(* This version of the block is self contained. Minimizes wiring.*)
FUNCTION_BLOCK FB_ExampleDeviceSM_DB
VAR_INPUT
	cBase: UDINT;
	iDBID:UDINT;
	sDBNetId: STRING;
	sDeviceID: STRING;
END_VAR
VAR_OUTPUT
END_VAR
VAR_IN_OUT
	fbArbiter : FB_Arbiter;
	fbFastFaultOutput	:	FB_HardwareFFOutput;
END_VAR
VAR
	stDevice	:	ST_Device;
	fbGovernor	:	FB_LinearGovernor;
	mcPower	:	MC_Power;
	mcStop: MC_Stop;
	mcAbsolute	:	MC_MoveAbsolute;
	fbBPTM	:	BeamParameterTransitionManager;
	xStartMove: BOOL;
	
	stCheckState: ST_DeviceState;
	stTargetState	:	ST_DeviceState; //Target device state
	fbDBClient:FB_MySQL_Client;
	bInitReady: BOOL :=FALSE;
	//aStateTable : ARRAY[1..PMPS_GVL.MAX_DEVICE_STATES] OF ST_DeviceStateTable;

END_VAR
VAR PERSISTENT
	nLastActiveState	:	UDINT;
END_VAR

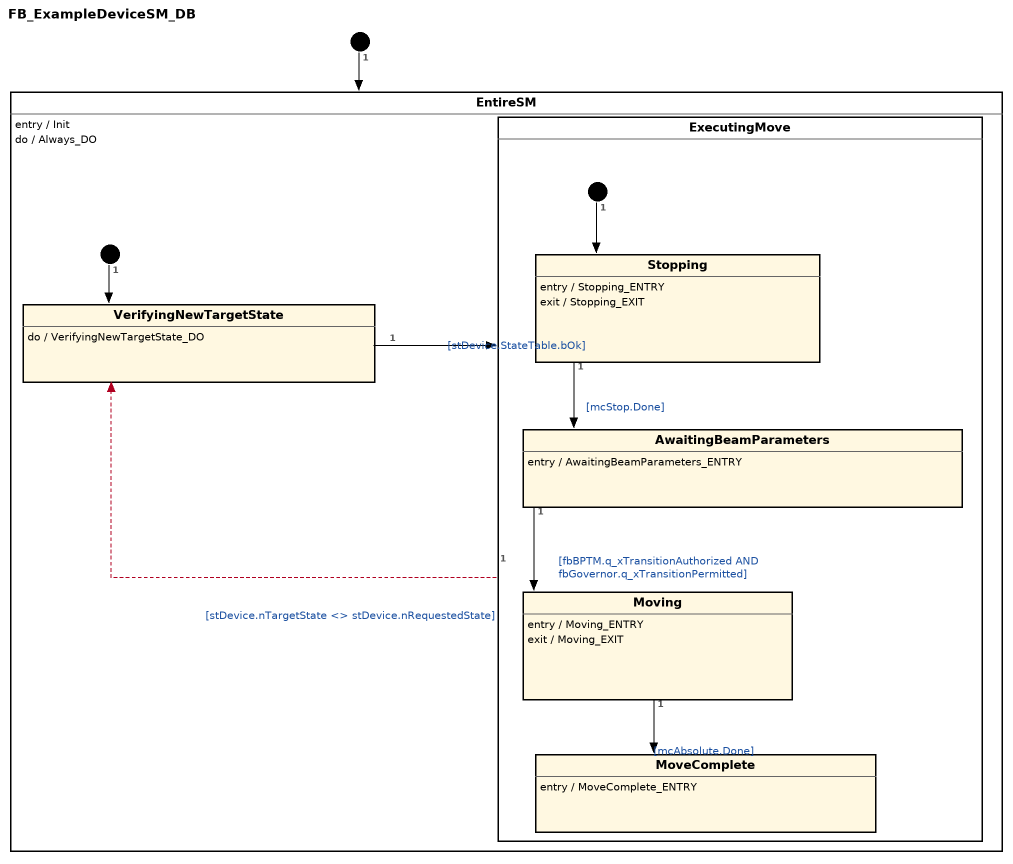
STATECHART FB_ExampleDeviceSM_DB  // abortable
    START StartState3
    COMPOSITE STATE EntireSM
        entry / Init
        do / Always_DO
        START StartState1
        COMPOSITE STATE ExecutingMove
            START StartState2
            STATE Stopping
                entry / Stopping_ENTRY
                exit / Stopping_EXIT
            STATE AwaitingBeamParameters
                entry / AwaitingBeamParameters_ENTRY
            STATE Moving
                entry / Moving_ENTRY
                exit / Moving_EXIT
            STATE MoveComplete
                entry / MoveComplete_ENTRY
            StartState2 -> Stopping  // priority 1, on completion
            Stopping -> AwaitingBeamParameters [mcStop.Done] // priority 1, rising edge
            AwaitingBeamParameters -> Moving [fbBPTM.q_xTransitionAuthorized AND fbGovernor.q_xTransitionPermitted] // priority 1, rising edge
            Moving -> MoveComplete [mcAbsolute.Done] // priority 1, rising edge
        END_STATE
        STATE VerifyingNewTargetState
            do / VerifyingNewTargetState_DO
        StartState1 -> VerifyingNewTargetState  // priority 1, on completion
        ExecutingMove -> VerifyingNewTargetState [stDevice.nTargetState <> stDevice.nRequestedState] // priority 1, exception, rising edge
        VerifyingNewTargetState -> ExecutingMove [stDevice.StateTable.bOk] // priority 1
    END_STATE
    StartState3 -> EntireSM  // priority 1, on completion
END_STATECHART

ACTION Always_DO:
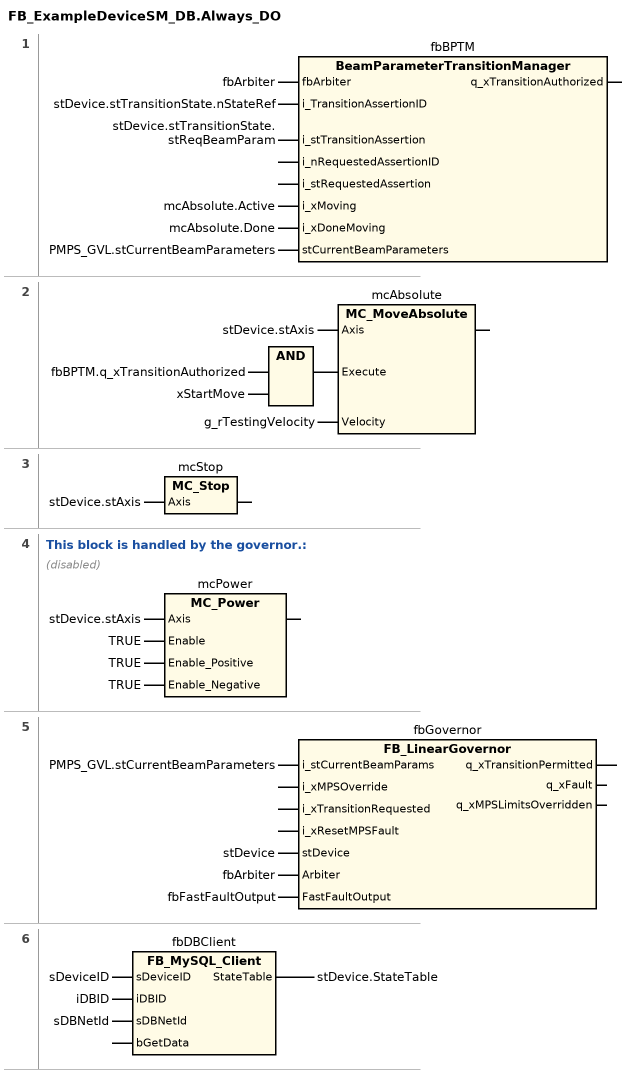
// NETWORK 1
fbBPTM(
    fbArbiter := fbArbiter,
    i_TransitionAssertionID := stDevice.stTransitionState.nStateRef,
    i_stTransitionAssertion := stDevice.stTransitionState.stReqBeamParam,
    i_xMoving := mcAbsolute.Active,
    i_xDoneMoving := mcAbsolute.Done,
    stCurrentBeamParameters := PMPS_GVL.stCurrentBeamParameters); // BeamParameterTransitionManager

// NETWORK 2
mcAbsolute(
    Axis := stDevice.stAxis,
    Execute := fbBPTM.q_xTransitionAuthorized AND xStartMove,
    Velocity := g_rTestingVelocity); // MC_MoveAbsolute

// NETWORK 3
mcStop(Axis := stDevice.stAxis); // MC_Stop

// NETWORK 4 (disabled)
// label: This block is handled by the governor.
// mcPower(Axis := stDevice.stAxis, Enable := TRUE, Enable_Positive := TRUE, Enable_Negative := TRUE); // MC_Power

// NETWORK 5
fbGovernor(
    i_stCurrentBeamParams := PMPS_GVL.stCurrentBeamParameters,
    stDevice := stDevice,
    Arbiter := fbArbiter,
    FastFaultOutput := fbFastFaultOutput); // FB_LinearGovernor

// NETWORK 6
fbDBClient(sDeviceID := sDeviceID, iDBID := iDBID, sDBNetId := sDBNetId); // FB_MySQL_Client
stDevice.StateTable := fbDBClient.StateTable;
END_ACTION

ACTION AwaitingBeamParameters_ENTRY:
fbBPTM.i_stRequestedAssertion := stTargetState.stReqBeamParam;
fbBPTM.i_nRequestedAssertionID := stTargetState.nStateRef;

//Tell the governor that we're trying to move.
fbGovernor.i_xTransitionRequested := TRUE;
END_ACTION

ACTION Init:
	
//Safe State
stDevice.nSafeState := cBase;
stDevice.nTransitionState := cBase+100;

//Initialize the State Table
stDevice.StateTable.A_Reset();
//Device State Table Instantiation
F_SetStateParams(
	nStateRef := stDevice.nSafeState,
	rPosition := 0,
	rTolerance := 10,
	stBeamParams := PMPS_GVL.cstFullBeam,
	Table := stDevice.StateTable
);
//Connect to DB and get state table data
fbDBClient.bGetData:= TRUE;//fbMySQL.nState:=400; 

stDevice.StateTable.A_Lookup(
		key := stDevice.nTransitionState,
		getValue => stDevice.stTransitionState
);
	
//Need an initialization routine for setting the active state
//Check if the device is at the last known state
//If the device is within the state boundaries, it's considered to be in that state
stDevice.StateTable.A_Lookup(key:= nLastActiveState);
IF stDevice.StateTable.bOk THEN
	stCheckState := stDevice.StateTable.getValue;
ELSE
	stCheckState := stDevice.stTransitionState; //This needs to be safer <TODO>
END_IF

IF stDevice.stAxis.NcToPlc.ActPos <= stCheckstate.rPosition + stCheckState.rTolerance AND
	stDevice.stAxis.NcToPlc.ActPos >= stCheckState.rPosition - stCheckState.rTolerance THEN
	stDevice.nActiveState := nLastActiveState;
ELSE
	stDevice.nActiveState := stDevice.nTransitionState;
END_IF

//Simulation Hardware Limit Switches
stDevice.i_xHiLim := TRUE;
stDevice.i_xLoLim := TRUE;
END_ACTION

ACTION Initialize:

END_ACTION

ACTION MoveComplete_ENTRY:
//Clear transition request
fbGovernor.i_xTransitionRequested := FALSE;
//Latch active state
stDevice.nActiveState := stDevice.nTargetState;
nLastActiveState := stDevice.nActiveState;
END_ACTION

ACTION Moving_ENTRY:
xStartMove := TRUE;
mcAbsolute.Position := stTargetState.rPosition;
END_ACTION

ACTION Moving_EXIT:
xStartMove := FALSE;
END_ACTION

ACTION NewMove_ENTRY:

END_ACTION

ACTION Stopping_ENTRY:
mcStop.Execute := TRUE;
END_ACTION

ACTION Stopping_EXIT:
mcStop.Execute := FALSE;
END_ACTION

ACTION VerifyingNewTargetState_DO:
stDevice.StateTable.A_Lookup(
	key := stDevice.nRequestedState
);

IF stDevice.StateTable.bOk THEN
	stTargetState := stDevice.StateTable.getValue;
	stDevice.nTargetState := stDevice.nRequestedState;
ELSE
	; //log ignored state/ generate an error? <TODO>
END_IF
END_ACTION

END_FUNCTION_BLOCK

(* stored: Version 1.1.0.1, ProductVersion 3.1.4022.18
   POU FB_ExampleDeviceSM_DB: Id {41eb4ad8-b23a-028e-1548-3249bc1b1092}, SpecialFunc None
   Action Always_DO: Id {8dada57c-e47d-076a-3d1f-0cbb1fb9477b}
   Action AwaitingBeamParameters_ENTRY: Id {087cc368-f96b-0b39-2d06-a053e4a69524}
   Action Init: Id {81eee3d4-8b32-00f4-245f-f0db40264a30}
   Action Initialize: Id {0a13b2bd-7481-00ef-20d2-9af33adb7b00}
   Action MoveComplete_ENTRY: Id {cf2b82ec-b223-0c17-28d6-f9dbc950d2fb}
   Action Moving_ENTRY: Id {00360884-3f7e-0a8d-1948-e19634d97ccf}
   Action Moving_EXIT: Id {aa4300cf-8347-07c7-296f-776cc26ad6ff}
   Action NewMove_ENTRY: Id {e4674221-3bea-0010-34c2-37ff37d217d1}
   Action Stopping_ENTRY: Id {7bfcb6d5-7cdd-0d99-1d92-5acc5401826f}
   Action Stopping_EXIT: Id {b083b1d1-574f-06f5-3fa2-6274116e7846}
   Action VerifyingNewTargetState_DO: Id {5920eaa2-9cfe-07b5-0033-20107a6678f2} *)
